FUNCTION_BLOCK handle
VAR_INPUT
END_VAR
VAR_OUTPUT
END_VAR
VAR
	i,j,k:INT;
	v_step		: LREAL;
	avg_window	: INT;
	avg_window_size : INT := 20;
	return_handoff_bypass : BOOL;

	act_hh		:	ARRAY[1..7] OF ARRAY [1..30] OF LREAL;
	pos_abs		:	LREAL;
	legacy_vel	:	LREAL;

	init_done : BOOL := FALSE;
	all_enabled : BOOL;
	all_powered : BOOL;
	has_axis_error : BOOL;
	hold_active : BOOL := FALSE;

	// 上位机通信看门狗。超时锁存后只能通过显式恢复握手解除。
	host_watchdog_timer : TON;
	host_last_session_id : UDINT := 0;
	host_last_heartbeat_sequence : UDINT := 0;
	host_heartbeat_seen : BOOL := FALSE;
	host_session_changed : BOOL;
	host_heartbeat_changed : BOOL;
	host_timeout_latched : BOOL := TRUE;
	host_timeout_prev : BOOL := FALSE;
	// 看门狗超时后锁存一次外部设定值保持位置。
	// 不能每拍把 Actual Position 回写为下一拍设定值，否则编码器微动会被回灌到 NC。
	host_hold_abs : ARRAY[1..7] OF LREAL;
	host_hold_captured : BOOL := FALSE;
	host_all_stopped : BOOL;
	host_return_stop_active : ARRAY[1..7] OF BOOL;
	host_return_stop_exec : ARRAY[1..7] OF BOOL;
	host_axis4_stop_active : BOOL := FALSE;
	fb_host_return_stop : ARRAY[1..7] OF MC_Stop;

	right_slimit : ARRAY[1..7] OF LREAL;
	rslimit_distance	: ARRAY[1..7] OF LREAL := [99.0, 0.0, 666.0, 0.0, 688.0, 688.0, 0.0];
	slimit_enable : ARRAY[1..7] OF BOOL := [TRUE, FALSE, FALSE, FALSE, TRUE, TRUE, FALSE];

	ext_setpoint_enabled : ARRAY[1..7] OF BOOL := [FALSE,FALSE,FALSE,FALSE,FALSE,FALSE,FALSE];
	spg_enable_exec	: ARRAY[1..7] OF BOOL;
	spg_disable_exec : ARRAY[1..7] OF BOOL;

	return_enable : ARRAY[1..7] OF BOOL := [TRUE, FALSE, FALSE, FALSE, TRUE, TRUE, FALSE];
	return_state : ARRAY[1..7] OF INT;
	return_exec : ARRAY[1..7] OF BOOL;
	return_target_abs : ARRAY[1..7] OF LREAL;
	return_velocity : ARRAY[1..7] OF LREAL;
	return_acc : ARRAY[1..7] OF LREAL;
	return_dec : ARRAY[1..7] OF LREAL;
	return_jerk : ARRAY[1..7] OF LREAL;
	return_finish_error : ARRAY[1..7] OF BOOL;
	return_cancelled : ARRAY[1..7] OF BOOL;
	return_error_id_pending : ARRAY[1..7] OF UDINT;
	fb_return_move_abs : ARRAY[1..7] OF MC_MoveAbsolute;

	axis4_manual_state : INT := 0;
	axis4_request_dir_now : INT := 0;
	axis4_requested_dir : INT := 0;
	axis4_pending_dir : INT := 0;
	axis4_move_exec : BOOL := FALSE;
	axis4_stop_exec : BOOL := FALSE;
	axis4_finish_error : BOOL := FALSE;
	axis4_error_id_pending : UDINT := 0;
	axis4_manual_velocity : LREAL := 30;
	axis4_manual_acc : LREAL := 100;
	axis4_manual_dec : LREAL := 100;
	axis4_manual_jerk : LREAL := 500.0;
	axis4_manual_direction : MC_Direction := MC_Direction.MC_Positive_Direction;
	fb_axis4_move_velocity : MC_MoveVelocity;
	fb_axis4_stop : MC_Stop;
	ramp_counter: ARRAY[1..7] OF INT;
	act_h_prev : ARRAY[1..7] OF LREAL;

	traj_pos     : ARRAY[1..7] OF LREAL;
	traj_vel     : ARRAY[1..7] OF LREAL;
	traj_acc     : ARRAY[1..7] OF LREAL;
	acc_raw      : LREAL;

	traj_wn      : LREAL := 60.0;
	traj_vmax    : ARRAY[1..7] OF LREAL := [80, 0, 0, 0, 80, 80, 0];
	traj_amax    : ARRAY[1..7] OF LREAL := [2000, 0, 0, 0, 2000, 2000, 0];
	traj_enable  : ARRAY[1..7] OF BOOL := [TRUE, FALSE, FALSE, FALSE, TRUE, TRUE, FALSE];
	pd_mode : USINT;
	pd_state : USINT;
	pd_last_state : USINT;
	pd_last_sync : USINT;
	pd_step : USINT;
	pd_axis : INT := 1;
	pd_active : ARRAY[1..7] OF BOOL;
	pd_req : ARRAY[1..7] OF BOOL;
	pd_moved : ARRAY[1..7] OF BOOL;
	pd_ref : ARRAY[1..7] OF LREAL;
	pd_target : ARRAY[1..7] OF LREAL;
	pd_forward : ST_AxisPlannedReturnCmd;
	pd_return : ST_AxisPlannedReturnCmd;
	pd_release_wait, pd_reclamp_wait, pd_release_lead, pd_reclamp_lead : TIME;
	pd_open2, pd_close2, pd_open4, pd_close4 : WORD;
	pd_coupling : BOOL;
	pd_ready : BOOL;
	pd_fault : BOOL;
	pd_all_done : BOOL;
	pd_anchor1, pd_anchor5, pd_anchor6, pd_input1, pd_input2 : LREAL;
	pd_baseline_timer, pd_release_timer, pd_reclamp_timer : TON;
	pd_release_lead_timer, pd_reclamp_lead_timer : TON;
	rec_block : INT := 1;
	rec_index : INT;
	rec_sample : UDINT;
	rec_sequence : UDINT;
	rec_was_active : BOOL;
	rec_capture : BOOL;
	rec_time : ULINT;
	zero_index : UINT;
	zero_force, zero_sum, zero_square, zero_mean, zero_std : ARRAY[1..4] OF LREAL;
END_VAR

host_session_changed := G.host_session_id <> host_last_session_id;
host_heartbeat_changed := host_session_changed OR
	(G.host_heartbeat_sequence <> host_last_heartbeat_sequence);

IF host_session_changed THEN
	// 非零会话发生变化表示新的上位机接管，必须重新完成恢复握手。
	IF host_last_session_id <> 0 THEN
		host_timeout_latched := TRUE;
	END_IF
	host_last_session_id := G.host_session_id;
END_IF

IF host_heartbeat_changed THEN
	host_last_heartbeat_sequence := G.host_heartbeat_sequence;
END_IF

host_heartbeat_seen := G.host_session_id <> 0;
// 心跳变化的扫描周期将 TON 复位；序号连续 100 ms 不变化才判定通信超时。
host_watchdog_timer(
	IN:=host_heartbeat_seen AND NOT host_heartbeat_changed,
	PT:=T#100MS
);
IF (NOT host_heartbeat_seen) OR host_watchdog_timer.Q THEN
	host_timeout_latched := TRUE;
END_IF
G.host_comm_timeout := host_timeout_latched;

IF G.handle_reinit_req THEN
	init_done := FALSE;
	G.handle_reinit_done := FALSE;
	G.handle_reinit_req := FALSE;
	G.estop_hold_req := TRUE;

	FOR i:=1 TO 7 DO
		ext_setpoint_enabled[i] := FALSE;
		spg_enable_exec[i] := FALSE;
		spg_disable_exec[i] := FALSE;
		return_state[i] := 0;
		return_exec[i] := FALSE;
		return_finish_error[i] := FALSE;
		return_cancelled[i] := FALSE;
		return_error_id_pending[i] := 0;
		host_return_stop_active[i] := FALSE;
		host_return_stop_exec[i] := FALSE;
		traj_pos[i] := 0.0;
		traj_vel[i] := 0.0;
		traj_acc[i] := 0.0;
		host_hold_abs[i] := 0.0;
		G.return_cmd[i].Req := FALSE;
		G.return_cmd[i].Busy := FALSE;
		G.return_cmd[i].Done := FALSE;
		G.return_cmd[i].Error := FALSE;
		G.return_cmd[i].ErrorId := 0;
	END_FOR
	host_hold_captured := FALSE;
	host_timeout_prev := FALSE;

	axis4_manual_state := 0;
	axis4_request_dir_now := 0;
	axis4_requested_dir := 0;
	axis4_pending_dir := 0;
	axis4_move_exec := FALSE;
	axis4_stop_exec := FALSE;
	axis4_finish_error := FALSE;
	axis4_error_id_pending := 0;
	G.axis4_fwd_req := FALSE;
	G.axis4_rev_req := FALSE;
	G.axis4_manual_busy := FALSE;
	G.axis4_manual_done := FALSE;
	G.axis4_manual_error := FALSE;
	G.axis4_manual_error_id := 0;
END_IF

IF NOT init_done THEN
	G.estop_hold_req := TRUE;
	G.power_[3].Enable := FALSE;
	all_enabled := TRUE;
	FOR i:=1 TO 7 DO
		IF i = 3 THEN
			G.SetPointGenEnable[i](Axis:=G.axis[i], Execute:=FALSE);
		ELSE
			G.SetPointGenEnable[i](Axis:=G.axis[i], Execute:=TRUE);
			IF NOT G.SetPointGenEnable[i].Done THEN
				all_enabled := FALSE;
			END_IF
		END_IF
	END_FOR
	
	IF all_enabled THEN
		FOR j:=1 TO 7 DO
			G.Act_pos[j] := G.axis[j].NcToPlc.ActPos - G.init_pos[j];
			G.act_pos_from_left[j] := G.axis[j].NcToPlc.ActPos - G.leftlimit[j];
			G.ref_slow[j] := G.Act_pos[j];
			G.act_h[j] := G.Act_pos[j];
			G.act_hf[j] := G.Act_pos[j];
			G.refer[j] := G.Act_pos[j];
			G.refer_from_left[j] := G.act_pos_from_left[j];
			ext_setpoint_enabled[j] := j <> 3;

			FOR k:=1 TO 30 DO
				act_hh[j][k] := G.Act_pos[j];
			END_FOR
			act_h_prev[j] := G.Act_pos[j];
			traj_pos[j] := G.Act_pos[j];
			traj_vel[j] := 0.0;
			traj_acc[j] := 0.0;
			IF slimit_enable[j] THEN
				right_slimit[j] := G.leftlimit[j] + rslimit_distance[j];
			END_IF
			G.return_cmd[j].Busy := FALSE;
			G.return_cmd[j].Done := FALSE;
			G.return_cmd[j].Error := FALSE;
			G.return_cmd[j].ErrorId := 0;
		END_FOR

		G.axis4_manual_busy := FALSE;
		G.axis4_manual_done := FALSE;
		G.axis4_manual_error := FALSE;
		G.axis4_manual_error_id := 0;

		init_done := TRUE;
		// 通信超时未解除时不提前确认恢复；正式握手后会再次进入本初始化流程。
		G.handle_reinit_done := NOT G.host_comm_timeout;
	END_IF
	RETURN;
END_IF

G.estop_hold_req := FALSE;
G.power_[3].Enable := FALSE;
G.power_[5].Enable := TRUE;

all_powered := TRUE;
FOR i:=1 TO 7 DO
	IF i <> 3 AND NOT (G.program_test_mode = 1 AND i = 5) AND NOT G.power_output[i].Done THEN
		all_powered := FALSE;
		EXIT;
	END_IF
END_FOR

has_axis_error := FALSE;
FOR i:=1 TO 7 DO
	IF i = 3 OR (G.program_test_mode = 1 AND i = 5) THEN
		CONTINUE;
	END_IF
	IF G.axis[i].Status.Error OR G.power_output[i].Error OR G.reset_output[i].Error THEN
		has_axis_error := TRUE;
		EXIT;
	END_IF
END_FOR


IF (NOT all_powered) OR has_axis_error OR G.host_comm_timeout THEN
	pd_fault := TRUE;
	ProgramDelivery();
	ProgramRecord();
END_IF

IF NOT all_powered THEN
	G.estop_hold_req := TRUE;
	hold_active := TRUE;
	FOR j:=1 TO 7 DO
		G.Act_pos[j] := G.axis[j].NcToPlc.ActPos - G.init_pos[j];
		G.act_pos_from_left[j] := G.axis[j].NcToPlc.ActPos - G.leftlimit[j];
		G.refer[j] := G.Act_pos[j];
		G.ref_slow[j] := G.Act_pos[j];
		G.act_h[j] := G.Act_pos[j];
		G.act_hf[j] := G.Act_pos[j];
		G.refer_from_left[j] := G.act_pos_from_left[j];
		FOR k:=1 TO 30 DO
			act_hh[j][k] := G.Act_pos[j];
		END_FOR
		act_h_prev[j] := G.Act_pos[j];
		traj_pos[j] := G.Act_pos[j];
		traj_vel[j] := 0.0;
		traj_acc[j] := 0.0;
	END_FOR
	IF has_axis_error THEN
		G.gen_state := _err;
	END_IF
	RETURN;
END_IF

IF hold_active THEN
	hold_active := FALSE;
	G.handle_reinit_req := TRUE;
	G.estop_hold_req := TRUE;
	IF has_axis_error THEN
		G.gen_state := _err;
	END_IF
	RETURN;
END_IF

IF has_axis_error THEN
	G.estop_hold_req := TRUE;
	G.gen_state := _err;
	RETURN;
END_IF

IF G.host_comm_timeout THEN
	G.estop_hold_req := TRUE;
	G.handle_reinit_done := FALSE;

	IF (NOT host_timeout_prev) OR (NOT host_hold_captured) THEN
		// 仅在进入超时保持时采样一次。之后始终维持同一绝对位置，
		// 避免 Actual -> Set Position 的逐周期回灌导致低频来回摆动。
		FOR i:=1 TO 7 DO
			host_hold_abs[i] := G.axis[i].NcToPlc.ActPos;
		END_FOR
		host_hold_captured := TRUE;
	END_IF

	IF NOT host_timeout_prev THEN
		// 仅捕获超时发生时已经在运行的独立运动，禁止恢复后自动续跑。
		FOR i:=1 TO 7 DO
			host_return_stop_active[i] :=
				(return_state[i] <> 0) OR G.return_cmd[i].Busy OR fb_return_move_abs[i].Busy;
			host_return_stop_exec[i] := FALSE;
		END_FOR
		host_axis4_stop_active := (axis4_manual_state <> 0) OR fb_axis4_move_velocity.Busy;
	END_IF

	// 超时期间持续清除运动请求，避免上位机重连时把旧请求重新送入状态机。
	G.axis1_fast_return := FALSE;
	G.axis6_fast_retract := FALSE;
	G.axis4_fwd_req := FALSE;
	G.axis4_rev_req := FALSE;
	G.startup_smoothing_bypass := FALSE;
	axis4_move_exec := FALSE;
	host_all_stopped := TRUE;

	FOR i:=1 TO 7 DO
		spg_enable_exec[i] := FALSE;
		spg_disable_exec[i] := FALSE;
		return_exec[i] := FALSE;
		G.return_cmd[i].Req := FALSE;
		G.return_cmd[i].Done := FALSE;

		// 实际位置仍实时刷新用于诊断；外部参考始终保持超时边沿的锁存位置。
		G.Act_pos[i] := G.axis[i].NcToPlc.ActPos - G.init_pos[i];
		G.act_pos_from_left[i] := G.axis[i].NcToPlc.ActPos - G.leftlimit[i];
		G.refer[i] := host_hold_abs[i] - G.init_pos[i];
		G.ref_slow[i] := G.refer[i];
		G.act_h[i] := G.refer[i];
		G.act_hf[i] := G.refer[i];
		G.refer_from_left[i] := host_hold_abs[i] - G.leftlimit[i];
		FOR k:=1 TO 30 DO
			act_hh[i][k] := G.refer[i];
		END_FOR
		act_h_prev[i] := G.refer[i];
		traj_pos[i] := G.refer[i];
		traj_vel[i] := 0.0;
		traj_acc[i] := 0.0;

		IF host_return_stop_active[i] THEN
			IF fb_host_return_stop[i].Done THEN
				host_return_stop_exec[i] := FALSE;
				host_return_stop_active[i] := FALSE;
			ELSIF fb_host_return_stop[i].Error THEN
				// 拉低一个扫描周期清除错误，下一周期继续尝试受控停止。
				host_return_stop_exec[i] := FALSE;
				host_all_stopped := FALSE;
			ELSE
				host_return_stop_exec[i] := TRUE;
				host_all_stopped := FALSE;
			END_IF
		ELSE
			host_return_stop_exec[i] := FALSE;
		END_IF
		G.return_cmd[i].Busy := host_return_stop_active[i];

		IF ext_setpoint_enabled[i] THEN
			MC_ExtSetPointGenFeed(
				Position:=host_hold_abs[i],
				Velocity:=0.0,
				Acceleration:=0.0,
				Direction:=1,
				Axis:=G.axis[i]);
		END_IF

		// 所有运动功能块在看门狗分支中仍保持每扫描调用。
		G.SetPointGenEnable[i](Axis:=G.axis[i], Execute:=FALSE);
		G.SetPointGenDisable[i](Axis:=G.axis[i], Execute:=FALSE);
		fb_return_move_abs[i](
			Axis:=G.axis[i],
			Position:=return_target_abs[i],
			Velocity:=return_velocity[i],
			Acceleration:=return_acc[i],
			Deceleration:=return_dec[i],
			Jerk:=return_jerk[i],
			Execute:=FALSE
		);
		fb_host_return_stop[i](
			Axis:=G.axis[i],
			Execute:=host_return_stop_exec[i],
			Deceleration:=100.0,
			Jerk:=500.0
		);
	END_FOR

	IF host_axis4_stop_active THEN
		IF fb_axis4_stop.Done THEN
			axis4_stop_exec := FALSE;
			host_axis4_stop_active := FALSE;
		ELSIF fb_axis4_stop.Error THEN
			// 拉低一个扫描周期清除错误，下一周期继续尝试受控停止。
			axis4_stop_exec := FALSE;
			host_all_stopped := FALSE;
		ELSE
			axis4_stop_exec := TRUE;
			host_all_stopped := FALSE;
		END_IF
	ELSE
		axis4_stop_exec := FALSE;
	END_IF
	G.axis4_manual_busy := host_axis4_stop_active;
	G.axis4_manual_done := FALSE;

	fb_axis4_move_velocity(
		Axis:=G.axis[4],
		Execute:=FALSE,
		Velocity:=axis4_manual_velocity,
		Acceleration:=axis4_manual_acc,
		Deceleration:=axis4_manual_dec,
		Jerk:=axis4_manual_jerk,
		Direction:=axis4_manual_direction
	);
	fb_axis4_stop(
		Axis:=G.axis[4],
		Execute:=axis4_stop_exec,
		Deceleration:=axis4_manual_dec,
		Jerk:=axis4_manual_jerk
	);

	// 清请求并解除超时即为 PLC 对恢复请求的确认；随后复用既有重初始化流程。
	IF G.host_recover_req AND host_heartbeat_seen AND
		(NOT host_watchdog_timer.Q) AND host_all_stopped THEN
		host_timeout_latched := FALSE;
		G.host_comm_timeout := FALSE;
		G.host_recover_req := FALSE;
		G.handle_reinit_req := TRUE;
	END_IF

	host_timeout_prev := G.host_comm_timeout;
	RETURN;
END_IF

host_timeout_prev := FALSE;
host_hold_captured := FALSE;
// 非超时状态收到的恢复请求没有业务含义，清除以免成为下一次超时的陈旧握手。
G.host_recover_req := FALSE;

pd_fault := FALSE;
ProgramDelivery();
ProgramRecord();

IF G.cylinder5_press_req THEN
	G.cylinder5_value := 0;
ELSE
	G.cylinder5_value := 2000;
END_IF

FOR i:=1 TO 7 DO
	spg_enable_exec[i] := FALSE;
	spg_disable_exec[i] := FALSE;
	return_exec[i] := FALSE;
END_FOR
axis4_move_exec := FALSE;
axis4_stop_exec := FALSE;

FOR j:=1 TO 7 DO
	G.Act_pos[j] := G.axis[j].NcToPlc.ActPos - G.init_pos[j];
	G.act_pos_from_left[j] := G.axis[j].NcToPlc.ActPos - G.leftlimit[j];
	G.refer_from_left[j] := (G.refer[j] + G.init_pos[j]) - G.leftlimit[j];

	v_step := G.v_limit[j];
	// 回退接管旁路：回退 Busy 期间跳过斜坡/均值，避免回退末端重新进入慢链路
	return_handoff_bypass := ((j = 1) AND (G.axis1_fast_return OR G.return_cmd[1].Busy))
		OR ((j = 6) AND (G.axis6_fast_retract OR G.return_cmd[6].Busy));
	IF return_handoff_bypass THEN
		avg_window := 1;
		ramp_counter[j] := 0;
	ELSE
		ramp_counter[j] := MIN(ramp_counter[j] + 1, avg_window_size);
		avg_window := MAX(1, ramp_counter[j]);
	END_IF

	FOR k:=2 TO 20 DO
		act_hh[j][22-k] := act_hh[j][21-k];
	END_FOR

	IF slimit_enable[j] THEN
		IF (G.axis[j].NcToPlc.ActPos >= right_slimit[j]) AND (G.refer[j] > G.ref_slow[j]) THEN
			G.refer[j] := G.ref_slow[j];
		END_IF
	END_IF

	IF return_handoff_bypass THEN
		G.ref_slow[j] := G.refer[j];
	ELSIF (G.refer[j] - G.ref_slow[j]) > v_step THEN
		G.ref_slow[j] := G.ref_slow[j] + v_step;
	ELSIF (G.refer[j] - G.ref_slow[j]) < -v_step THEN
		G.ref_slow[j] := G.ref_slow[j] - v_step;
	ELSE
		G.ref_slow[j] := G.refer[j];
	END_IF

	IF return_handoff_bypass THEN
		FOR i:=1 TO 20 DO
			act_hh[j][i] := G.ref_slow[j];
		END_FOR
		G.act_h[j] := G.ref_slow[j];
	ELSE
		act_hh[j][1] := G.ref_slow[j];
		G.act_h[j] := 0;
		FOR i:=1 TO avg_window DO
			G.act_h[j] := G.act_h[j] + act_hh[j][i] / TO_LREAL(avg_window);
		END_FOR
	END_IF

	IF traj_enable[j] AND NOT return_handoff_bypass AND NOT G.startup_smoothing_bypass THEN
		acc_raw := traj_wn * traj_wn * (G.refer[j] - traj_pos[j]) - 2.0 * traj_wn * traj_vel[j];
		IF acc_raw > traj_amax[j] THEN
			acc_raw := traj_amax[j];
		ELSIF acc_raw < -traj_amax[j] THEN
			acc_raw := -traj_amax[j];
		END_IF
		traj_acc[j] := acc_raw;
		traj_vel[j] := traj_vel[j] + 0.001 * traj_acc[j];
		IF traj_vel[j] > traj_vmax[j] THEN
			traj_vel[j] := traj_vmax[j];
		ELSIF traj_vel[j] < -traj_vmax[j] THEN
			traj_vel[j] := -traj_vmax[j];
		END_IF
		traj_pos[j] := traj_pos[j] + 0.001 * traj_vel[j];
		IF ABS(G.refer[j] - traj_pos[j]) < 0.001 AND ABS(traj_vel[j]) < 0.01 THEN
			traj_pos[j] := G.refer[j];
			traj_vel[j] := 0.0;
			traj_acc[j] := 0.0;
		END_IF
	ELSE
		traj_pos[j] := G.act_h[j];
		traj_vel[j] := 0.0;
		traj_acc[j] := 0.0;
	END_IF
END_FOR

FOR i:=1 TO 7 DO
	IF NOT return_enable[i] AND NOT ((pd_mode <> 0) AND ((i = 2) OR (i = 7))) THEN
		CONTINUE;
	END_IF

	IF return_state[i] = 0 THEN
		G.return_cmd[i].Busy := FALSE;
		host_return_stop_active[i] := FALSE;
		host_return_stop_exec[i] := FALSE;
		IF NOT G.return_cmd[i].Req THEN
			G.return_cmd[i].Done := FALSE;
			G.return_cmd[i].Error := FALSE;
			G.return_cmd[i].ErrorId := 0;
			return_finish_error[i] := FALSE;
			return_cancelled[i] := FALSE;
			return_error_id_pending[i] := 0;
		ELSIF (NOT G.return_cmd[i].Done) AND (NOT G.return_cmd[i].Error) THEN
			// Req 由上位机在完整写入参数后最后置位；此处只锁存一次，
			// 本次 MC_MoveAbsolute 后续不再直接读取可被 ADS 改写的命令参数。
			return_target_abs[i] := G.return_cmd[i].TargetAbs;
			return_velocity[i] := G.return_cmd[i].Velocity;
			return_acc[i] := G.return_cmd[i].Acc;
			return_dec[i] := G.return_cmd[i].Dec;
			return_jerk[i] := G.return_cmd[i].Jerk;
			return_cancelled[i] := FALSE;
			return_state[i] := 10;
		END_IF
	END_IF

	// 上位机在任何尚未完成的阶段撤销请求时，都先受控停止轴。
	// return_cancelled防止状态40复用30/31收尾后因Req仍为FALSE再次进入停止环。
	IF ((return_state[i] = 10) OR (return_state[i] = 20) OR
		(return_state[i] = 30) OR (return_state[i] = 31)) AND
		(NOT G.return_cmd[i].Req) AND (NOT return_cancelled[i]) THEN
		return_exec[i] := FALSE;
		spg_enable_exec[i] := FALSE;
		spg_disable_exec[i] := FALSE;
		return_cancelled[i] := TRUE;
		host_return_stop_active[i] := TRUE;
		// 清除上一次执行沿；状态 40 首次处理时不会采信旧的 Done/Error。
		host_return_stop_exec[i] := FALSE;
		G.return_cmd[i].Done := FALSE;
		G.return_cmd[i].Error := FALSE;
		G.return_cmd[i].ErrorId := 0;
		return_state[i] := 40;
	END_IF

	CASE return_state[i] OF
	10:
		G.return_cmd[i].Busy := TRUE;
		spg_disable_exec[i] := TRUE;
		IF G.SetPointGenDisable[i].Done OR NOT G.SetPointGenDisable[i].Enabled THEN
			ext_setpoint_enabled[i] := FALSE;
			return_state[i] := 20;
		END_IF

	20:
		G.return_cmd[i].Busy := TRUE;
		return_exec[i] := TRUE;
		G.refer_from_left[i] := return_target_abs[i] - G.leftlimit[i];

		IF fb_return_move_abs[i].Done OR
		   ((NOT fb_return_move_abs[i].Busy) AND (ABS(G.axis[i].NcToPlc.ActPos - return_target_abs[i]) <= 0.05)) THEN
			return_finish_error[i] := FALSE;
			return_error_id_pending[i] := 0;
			return_state[i] := 30;
		ELSIF fb_return_move_abs[i].Error OR fb_return_move_abs[i].CommandAborted THEN
			return_finish_error[i] := TRUE;
			return_error_id_pending[i] := fb_return_move_abs[i].ErrorID;
			return_state[i] := 30;
		END_IF

	30:
		G.return_cmd[i].Busy := TRUE;
		IF ABS(G.axis[i].NcToPlc.ActVelo) <= 0.5 THEN
			G.Act_pos[i] := G.axis[i].NcToPlc.ActPos - G.init_pos[i];
			G.act_pos_from_left[i] := G.axis[i].NcToPlc.ActPos - G.leftlimit[i];
			G.refer[i] := G.Act_pos[i];
			G.ref_slow[i] := G.Act_pos[i];
			G.act_h[i] := G.Act_pos[i];
			G.act_hf[i] := G.Act_pos[i];
			G.refer_from_left[i] := G.act_pos_from_left[i];
			FOR k:=1 TO 30 DO
				act_hh[i][k] := G.Act_pos[i];
			END_FOR
			act_h_prev[i] := G.Act_pos[i];
			traj_pos[i] := G.Act_pos[i];
			traj_vel[i] := 0.0;
			traj_acc[i] := 0.0;
			// 先留出一个完整 PLC 扫描周期预送当前设定值，再重新使能外部设定值发生器。
			return_state[i] := 31;
		END_IF

	31:
		G.return_cmd[i].Busy := TRUE;
		spg_enable_exec[i] := TRUE;
		IF G.SetPointGenEnable[i].Done THEN
			ext_setpoint_enabled[i] := TRUE;
			G.return_cmd[i].Busy := FALSE;
			IF return_finish_error[i] THEN
				G.return_cmd[i].Done := FALSE;
				G.return_cmd[i].Error := TRUE;
				G.return_cmd[i].ErrorId := return_error_id_pending[i];
			ELSIF return_cancelled[i] THEN
				// 主动取消只表示已经安全停稳，不把取消伪装成原计划动作成功完成。
				G.return_cmd[i].Done := FALSE;
				G.return_cmd[i].Error := FALSE;
				G.return_cmd[i].ErrorId := 0;
			ELSE
				G.return_cmd[i].Done := TRUE;
				G.return_cmd[i].Error := FALSE;
				G.return_cmd[i].ErrorId := 0;
			END_IF
			return_finish_error[i] := FALSE;
			return_cancelled[i] := FALSE;
			return_error_id_pending[i] := 0;
			return_state[i] := 0;
		END_IF

	40:
		G.return_cmd[i].Busy := TRUE;
		G.return_cmd[i].Done := FALSE;
		return_exec[i] := FALSE;
		spg_enable_exec[i] := FALSE;
		spg_disable_exec[i] := FALSE;
		// 状态40仍以实际停稳为退出条件。若原运动或此前的MC_Stop已经报错，
		// 在继续受控停止期间保持错误对上位机可见，不能用Busy掩盖故障。
		IF return_finish_error[i] THEN
			G.return_cmd[i].Error := TRUE;
			G.return_cmd[i].ErrorId := return_error_id_pending[i];
		END_IF

		IF host_return_stop_exec[i] THEN
			IF fb_host_return_stop[i].Done THEN
				// 停稳后释放 MC_Stop，并复用状态 30/31 按实际位置重建和恢复外部设定值。
				host_return_stop_exec[i] := FALSE;
				host_return_stop_active[i] := FALSE;
				return_state[i] := 30;
			ELSIF fb_host_return_stop[i].Error THEN
				// 原运动错误优先；否则锁存首次MC_Stop错误并立即通知上位机。
				// Busy和停止任务保持有效，Execute拉低一拍后仍继续尝试受控停止，
				// 只有真实Done才能进入位置重建，绝不把停止失败伪装成完成。
				IF NOT return_finish_error[i] THEN
					return_finish_error[i] := TRUE;
					return_error_id_pending[i] := fb_host_return_stop[i].ErrorID;
				END_IF
				G.return_cmd[i].Error := TRUE;
				G.return_cmd[i].ErrorId := return_error_id_pending[i];
				host_return_stop_exec[i] := FALSE;
			END_IF
		ELSIF NOT fb_host_return_stop[i].Error THEN
			// 首次进入或错误已由低电平清除后，启动（或重试）受控停止。
			host_return_stop_exec[i] := TRUE;
		END_IF
	END_CASE
END_FOR

axis4_request_dir_now := 0;
IF G.axis4_fwd_req AND NOT G.axis4_rev_req THEN
	axis4_request_dir_now := 1;
ELSIF G.axis4_rev_req AND NOT G.axis4_fwd_req THEN
	axis4_request_dir_now := -1;
END_IF

IF axis4_manual_state = 0 THEN
	G.axis4_manual_busy := FALSE;
	IF axis4_request_dir_now = 0 THEN
		G.axis4_manual_done := FALSE;
		G.axis4_manual_error := FALSE;
		G.axis4_manual_error_id := 0;
	ELSIF NOT G.axis4_manual_error THEN
		G.axis4_manual_done := FALSE;
		G.axis4_manual_error := FALSE;
		G.axis4_manual_error_id := 0;
		axis4_requested_dir := axis4_request_dir_now;
		axis4_pending_dir := 0;
		axis4_finish_error := FALSE;
		axis4_error_id_pending := 0;
		axis4_manual_state := 10;
	END_IF
END_IF

CASE axis4_manual_state OF
10:
	G.axis4_manual_busy := TRUE;
	spg_disable_exec[4] := TRUE;
	IF G.SetPointGenDisable[4].Done OR NOT G.SetPointGenDisable[4].Enabled THEN
		ext_setpoint_enabled[4] := FALSE;
		axis4_manual_state := 20;
	END_IF

20:
	G.axis4_manual_busy := TRUE;
	axis4_pending_dir := axis4_request_dir_now;
	IF axis4_requested_dir >= 0 THEN
		axis4_manual_direction := MC_Direction.MC_Positive_Direction;
	ELSE
		axis4_manual_direction := MC_Direction.MC_Negative_Direction;
	END_IF

	IF axis4_pending_dir = 0 THEN
		axis4_manual_state := 30;
	ELSIF axis4_pending_dir <> axis4_requested_dir THEN
		axis4_manual_state := 30;
	ELSE
		axis4_move_exec := TRUE;
	END_IF

	IF fb_axis4_move_velocity.Error OR fb_axis4_move_velocity.CommandAborted THEN
		axis4_finish_error := TRUE;
		axis4_error_id_pending := fb_axis4_move_velocity.ErrorID;
		G.axis4_manual_error_id := fb_axis4_move_velocity.ErrorID;
		axis4_pending_dir := 0;
		axis4_manual_state := 40;
	END_IF

30:
	G.axis4_manual_busy := TRUE;
	axis4_pending_dir := axis4_request_dir_now;
	axis4_stop_exec := TRUE;

	IF fb_axis4_stop.Error THEN
		axis4_finish_error := TRUE;
		axis4_error_id_pending := fb_axis4_stop.ErrorID;
		axis4_pending_dir := 0;
		axis4_manual_state := 39;
	ELSIF fb_axis4_stop.Done OR (ABS(G.axis[4].NcToPlc.ActVelo) <= 0.05) THEN
		IF axis4_pending_dir <> 0 THEN
			axis4_requested_dir := axis4_pending_dir;
			axis4_manual_state := 20;
		ELSE
			axis4_requested_dir := 0;
			axis4_manual_state := 39;
		END_IF
	END_IF

39:
G.axis4_manual_busy := TRUE;
// MC_Stop needs one cycle with Execute=FALSE before SetPointGenEnable can get a clean rising edge
axis4_manual_state := 40;
	
40:
	G.axis4_manual_busy := TRUE;
	G.Act_pos[4] := G.axis[4].NcToPlc.ActPos - G.init_pos[4];
	G.act_pos_from_left[4] := G.axis[4].NcToPlc.ActPos - G.leftlimit[4];
	G.refer[4] := G.Act_pos[4];
	G.ref_slow[4] := G.Act_pos[4];
	G.act_h[4] := G.Act_pos[4];
	G.act_hf[4] := G.Act_pos[4];
	G.refer_from_left[4] := G.act_pos_from_left[4];
	FOR k:=1 TO 30 DO
		act_hh[4][k] := G.Act_pos[4];
	END_FOR
	act_h_prev[4] := G.Act_pos[4];
	traj_pos[4] := G.Act_pos[4];
	traj_vel[4] := 0.0;
	traj_acc[4] := 0.0;
	spg_enable_exec[4] := TRUE;
	IF G.SetPointGenEnable[4].Done THEN
		ext_setpoint_enabled[4] := TRUE;
		G.axis4_manual_busy := FALSE;
		IF axis4_finish_error THEN
			G.axis4_manual_done := FALSE;
			G.axis4_manual_error := TRUE;
			G.axis4_manual_error_id := axis4_error_id_pending;
		ELSE
			G.axis4_manual_done := TRUE;
			G.axis4_manual_error := FALSE;
			G.axis4_manual_error_id := 0;
		END_IF
		axis4_finish_error := FALSE;
		axis4_error_id_pending := 0;
		axis4_manual_state := 0;
	END_IF
END_CASE

FOR i:=1 TO 7 DO
	IF i <> 3 AND G.power_output[i].Error THEN
		G.axis_Reset[i].Execute := TRUE;
	END_IF
END_FOR

FOR i:=1 TO 7 DO
	IF i = 3 THEN
		G.act_hf[i] := G.axis[i].NcToPlc.ActPos - G.init_pos[i];
	ELSIF ext_setpoint_enabled[i] OR (return_state[i] = 31) OR spg_enable_exec[i] THEN
		IF traj_enable[i] AND NOT G.startup_smoothing_bypass THEN
			pos_abs := traj_pos[i] + G.init_pos[i];
			MC_ExtSetPointGenFeed(
				Position     := pos_abs,
				Velocity     := traj_vel[i],
				Acceleration := traj_acc[i],
				Direction    := 1,
				Axis         := G.axis[i]);
		ELSE
			pos_abs := G.act_h[i] + G.init_pos[i];
			legacy_vel := (G.act_h[i] - act_h_prev[i]) / 0.001;
			MC_ExtSetPointGenFeed(
				Position     := pos_abs,
				Velocity     := legacy_vel,
				Acceleration := 0,
				Direction    := 1,
				Axis         := G.axis[i]);
		END_IF
		G.act_hf[i] := G.act_h[i];
	ELSE
		G.act_hf[i] := G.axis[i].NcToPlc.ActPos - G.init_pos[i];
	END_IF
	act_h_prev[i] := G.act_h[i];
END_FOR

FOR i:=1 TO 7 DO
	G.SetPointGenEnable[i](Axis:=G.axis[i], Execute:=spg_enable_exec[i]);
	G.SetPointGenDisable[i](Axis:=G.axis[i], Execute:=spg_disable_exec[i]);
	fb_return_move_abs[i](
		Axis:=G.axis[i],
		Position:=return_target_abs[i],
		Velocity:=return_velocity[i],
		Acceleration:=return_acc[i],
		Deceleration:=return_dec[i],
		Jerk:=return_jerk[i],
		Execute:=return_exec[i]
	);
	fb_host_return_stop[i](
		Axis:=G.axis[i],
		Execute:=host_return_stop_exec[i],
		Deceleration:=100.0,
		Jerk:=500.0
	);
END_FOR

fb_axis4_move_velocity(
	Axis:=G.axis[4],
	Execute:=axis4_move_exec,
	Velocity:=axis4_manual_velocity,
	Acceleration:=axis4_manual_acc,
	Deceleration:=axis4_manual_dec,
	Jerk:=axis4_manual_jerk,
	Direction:=axis4_manual_direction
);
fb_axis4_stop(
	Axis:=G.axis[4],
	Execute:=axis4_stop_exec,
	Deceleration:=axis4_manual_dec,
	Jerk:=axis4_manual_jerk
);

ACTION ProgramDelivery:


pd_all_done := TRUE;
FOR i := 1 TO 7 DO
	IF (return_state[i] <> 0) OR G.return_cmd[i].Busy THEN pd_all_done := FALSE; END_IF
END_FOR
IF G.program_test_mode <> pd_mode THEN
	IF ((pd_state = 0) OR (pd_state >= 10)) AND NOT G.program_test_setup_busy AND pd_all_done THEN
		pd_mode := G.program_test_mode;
		pd_state := 0;
		pd_step := 0;
		pd_ready := FALSE;
		G.program_test_setup_done := FALSE;
		G.program_test_status_error_id := 0;
		G.program_test_handle_cycle := 0;
		FOR i := 1 TO 7 DO
			pd_ref[i] := G.axis[i].NcToPlc.ActPos - G.init_pos[i];
		END_FOR
	ELSE
		G.program_test_mode := pd_mode;
		G.program_test_status_error_id := 16#7102;
	END_IF
END_IF
IF pd_mode = 0 THEN
	G.program_test_phase := 0;
	G.program_test_sync_state := 0;
	G.program_test_enable := FALSE;
	G.program_test_sample_arm := FALSE;
ELSE
pd_input1 := G.refer[1] + G.init_pos[1];
pd_input2 := G.refer[2] + G.init_pos[2];
IF pd_fault THEN
	pd_state := 12;
	G.program_test_status_error_id := 16#7305;
	IF NOT all_powered THEN
		G.program_test_error_source := 5;
	ELSIF has_axis_error THEN
		G.program_test_error_source := 6;
	ELSIF G.host_comm_timeout THEN
		G.program_test_error_source := 7;
	ELSE
		G.program_test_error_source := 0;
	END_IF
	G.program_test_error_axis := 0;
	G.program_test_error_phase := 0;
	G.program_test_error_target_abs := 0.0;
END_IF
IF G.program_test_abort_req THEN
	G.program_test_abort_req := FALSE;
	pd_state := 11;
END_IF
IF G.experiment_record_overflow THEN
	pd_state := 12;
	G.program_test_status_error_id := 16#7402;
END_IF
FOR i := 1 TO 7 DO
	IF (return_state[i] >= 30) OR (pd_req[i] AND G.return_cmd[i].Done) THEN
		pd_ref[i] := G.axis[i].NcToPlc.ActPos - G.init_pos[i];
	END_IF
	IF pd_req[i] AND G.return_cmd[i].Error THEN
		G.program_test_error_phase := pd_state;
		G.program_test_error_axis := INT_TO_USINT(i);
		G.program_test_error_target_abs := pd_target[i];
		G.program_test_status_error_id := G.return_cmd[i].ErrorId;
		IF G.program_test_status_error_id = 0 THEN
			G.program_test_status_error_id := 16#7306;
		END_IF
		pd_state := 12;
	END_IF
END_FOR
IF (pd_state >= 10) AND G.program_test_setup_req AND pd_all_done AND NOT pd_fault THEN
	pd_state := 0;
	pd_step := 0;
END_IF
IF (pd_state <> 0) AND (pd_state < 10) THEN G.program_test_setup_req := FALSE; END_IF
IF pd_state <> 2 THEN G.program_test_start_req := FALSE; END_IF

pd_baseline_timer(IN:=pd_state = 3, PT:=T#1S);
pd_release_timer(IN:=((pd_state = 1) AND (pd_step = 0)) OR ((pd_state = 5) AND (pd_step = 1)), PT:=pd_release_wait);
pd_reclamp_timer(IN:=(pd_state = 2) OR ((pd_state = 7) AND (pd_step = 1)), PT:=pd_reclamp_wait);
pd_release_lead_timer(IN:=(pd_state = 5) AND (pd_step = 0), PT:=pd_release_lead);
pd_reclamp_lead_timer(IN:=(pd_state = 7) AND (pd_step = 0), PT:=pd_reclamp_lead);
G.program_test_wait_action := 0;

CASE pd_state OF
0:
	IF G.program_test_setup_req AND NOT pd_fault THEN
		G.program_test_setup_req := FALSE;
		G.program_test_start_req := FALSE;
		G.program_test_status_error_id := 0;
		G.program_test_error_source := 0;
		G.program_test_error_axis := 0;
		G.program_test_error_phase := 0;
		G.program_test_error_target_abs := 0.0;
		G.program_test_cycle_index := 0;
		G.program_test_cycle_total := G.program_test_cycle_count;
		G.program_test_setup_done := FALSE;
		pd_ready := FALSE;
		pd_axis := 1;
		IF pd_mode = 2 THEN pd_axis := 6; END_IF
		IF NOT G.self_check_done OR NOT pd_all_done THEN
			G.program_test_status_error_id := 16#7201;
		ELSIF (pd_mode <> 1) AND (pd_mode <> 2) AND (pd_mode <> 4) THEN
			G.program_test_status_error_id := 16#7202;
		ELSIF G.program_test_cycle_count = 0 THEN
			G.program_test_status_error_id := 16#7203;
		ELSIF ((pd_mode = 1) OR (pd_mode = 4)) AND NOT
			((G.program_test_axis1_trigger_from_left_mm >= 0.0) AND
			(G.program_test_axis1_prepare_from_left_mm <= 96.0) AND
			(G.program_test_axis1_prepare_from_left_mm > G.program_test_axis1_trigger_from_left_mm)) THEN
			G.program_test_status_error_id := 16#7204;
		ELSIF (pd_mode = 2) AND NOT
			((G.program_test_axis5_from_left_mm >= 0.0) AND (G.program_test_axis5_from_left_mm <= 670.0) AND
			(G.program_test_axis6_prepare_from_left_mm <= 670.0) AND
			(G.program_test_axis6_trigger_from_left_mm >= 0.0) AND
			(G.program_test_axis6_prepare_from_left_mm > G.program_test_axis6_trigger_from_left_mm)) THEN
			G.program_test_status_error_id := 16#7204;
		ELSIF (pd_mode = 4) AND NOT
			((G.program_test_axis6_prepare_from_left_mm <= 670.0) AND
			(G.program_test_axis6_prepare_from_left_mm -
				UINT_TO_LREAL(G.program_test_cycle_count) *
				(G.program_test_axis1_prepare_from_left_mm - G.program_test_axis1_trigger_from_left_mm) >= 0.0)) THEN
			G.program_test_status_error_id := 16#7204;
		ELSIF NOT ((G.program_test_forward_velocity > 0.0) AND (G.program_test_forward_velocity < 1.0E100) AND
			(G.program_test_forward_acceleration > 0.0) AND (G.program_test_forward_acceleration < 1.0E100) AND
			(G.program_test_forward_deceleration > 0.0) AND (G.program_test_forward_deceleration < 1.0E100) AND
			(G.program_test_forward_jerk > 0.0) AND (G.program_test_forward_jerk < 1.0E100) AND
			(G.program_test_return_velocity > 0.0) AND (G.program_test_return_velocity < 1.0E100) AND
			(G.program_test_return_acceleration > 0.0) AND (G.program_test_return_acceleration < 1.0E100) AND
			(G.program_test_return_deceleration > 0.0) AND (G.program_test_return_deceleration < 1.0E100) AND
			(G.program_test_return_jerk > 0.0) AND (G.program_test_return_jerk < 1.0E100)) THEN
			G.program_test_status_error_id := 16#7205;
		ELSIF (G.program_test_release_wait_ms > 60000) OR (G.program_test_reclamp_wait_ms > 60000) OR
			(G.program_test_release_lead_ms > 60000) OR (G.program_test_reclamp_lead_ms > 60000) THEN
			G.program_test_status_error_id := 16#7207;
		END_IF
		IF G.program_test_status_error_id <> 0 THEN
			pd_state := 12;
		ELSE
			pd_forward.Velocity := G.program_test_forward_velocity;
			pd_forward.Acc := G.program_test_forward_acceleration;
			pd_forward.Dec := G.program_test_forward_deceleration;
			pd_forward.Jerk := G.program_test_forward_jerk;
			pd_return.Velocity := G.program_test_return_velocity;
			pd_return.Acc := G.program_test_return_acceleration;
			pd_return.Dec := G.program_test_return_deceleration;
			pd_return.Jerk := G.program_test_return_jerk;
			pd_release_wait := UDINT_TO_TIME(G.program_test_release_wait_ms);
			pd_reclamp_wait := UDINT_TO_TIME(G.program_test_reclamp_wait_ms);
			pd_release_lead := UDINT_TO_TIME(G.program_test_release_lead_ms);
			pd_reclamp_lead := UDINT_TO_TIME(G.program_test_reclamp_lead_ms);
			pd_open2 := MAX(WORD#5, G.program_test_cylinder2_open_word);
			pd_close2 := MAX(WORD#5, G.program_test_cylinder2_close_word);
			pd_open4 := MAX(WORD#5, G.program_test_cylinder4_open_word);
			pd_close4 := MAX(WORD#5, G.program_test_cylinder4_close_word);
			pd_coupling := G.program_test_cylinder1_coupling_enable OR (pd_mode = 4);
			IF pd_mode = 2 THEN pd_coupling := G.program_test_cylinder3_coupling_enable; END_IF
			G.program_test_target_axis1_abs := G.leftlimit[1] + G.program_test_axis1_prepare_from_left_mm;
			G.program_test_target_axis5_abs := G.leftlimit[5] + G.program_test_axis5_from_left_mm;
			G.program_test_target_axis6_abs := G.leftlimit[6] + G.program_test_axis6_prepare_from_left_mm;
			IF pd_mode = 4 THEN
				// 外源验证两条平移轴使用同一个手柄运动窗口。
				G.program_test_axis6_trigger_from_left_mm :=
					G.program_test_axis6_prepare_from_left_mm -
					(G.program_test_axis1_prepare_from_left_mm - G.program_test_axis1_trigger_from_left_mm);
			END_IF
			G.program_test_target_axis2_deg := G.program_test_axis2_angle_deg;
			G.program_test_target_axis7_deg := G.program_test_axis7_angle_deg;
			FOR i := 1 TO 7 DO
				pd_active[i] := FALSE;
				pd_req[i] := FALSE;
				pd_moved[i] := FALSE;
				pd_ref[i] := G.axis[i].NcToPlc.ActPos - G.init_pos[i];
				pd_target[i] := G.axis[i].NcToPlc.ActPos;
			END_FOR
			IF pd_mode = 2 THEN
				pd_active[5] := TRUE;
				pd_active[6] := TRUE;
				pd_active[7] := TRUE;
				pd_target[5] := G.program_test_target_axis5_abs;
				pd_target[6] := G.program_test_target_axis6_abs;
				pd_target[7] := G.program_test_target_axis7_deg;
				G.program_test_trigger_target_abs := G.leftlimit[6] + G.program_test_axis6_trigger_from_left_mm;
				G.program_test_return_target_abs := pd_target[6];
				G.cylinder3_value := 400;
				IF pd_coupling THEN G.cylinder3_value := 50; END_IF
				G.cylinder4_value := pd_open4;
			ELSE
				pd_active[1] := TRUE;
				pd_active[2] := TRUE;
				pd_target[1] := G.program_test_target_axis1_abs;
				pd_target[2] := G.program_test_target_axis2_deg;
				G.program_test_trigger_target_abs := G.leftlimit[1] + G.program_test_axis1_trigger_from_left_mm;
				G.program_test_return_target_abs := pd_target[1];
				G.cylinder1_value := 400;
				IF pd_coupling THEN G.cylinder1_value := 5; END_IF
				G.cylinder2_value := pd_open2;
			END_IF
			G.program_test_final_target_abs := G.program_test_return_target_abs - G.program_test_final_forward_distance_mm;
			IF pd_mode = 4 THEN
				pd_active[6] := TRUE;
				pd_active[7] := TRUE;
				pd_target[6] := G.program_test_target_axis6_abs;
				pd_target[7] := pd_target[2];
				G.program_test_target_axis7_deg := pd_target[2];
				G.program_test_final_target_abs := G.program_test_return_target_abs;
				G.cylinder3_value := 400;
				G.cylinder4_value := pd_open4;
			END_IF
			pd_state := 1;
		END_IF
	END_IF
1:
	G.program_test_wait_action := 1;
	IF (pd_step = 0) AND pd_release_timer.Q THEN
		FOR i := 1 TO 7 DO pd_req[i] := pd_active[i]; END_FOR
		pd_step := 1;
	END_IF
	IF pd_step = 1 THEN
		G.program_test_wait_action := 0;
		pd_all_done := TRUE;
		FOR i := 1 TO 7 DO
			IF pd_active[i] THEN
				IF G.return_cmd[i].Done THEN
					pd_moved[i] := TRUE;
					pd_req[i] := FALSE;
				END_IF
				IF NOT pd_moved[i] THEN pd_all_done := FALSE; END_IF
			END_IF
		END_FOR
		IF pd_all_done THEN pd_state := 2; END_IF
	END_IF
2:
	IF pd_axis = 1 THEN
		G.cylinder1_value := 400;
		G.cylinder2_value := pd_close2;
	ELSE
		G.cylinder3_value := 400;
		G.cylinder4_value := pd_close4;
	END_IF
	IF pd_mode = 4 THEN G.cylinder4_value := pd_close4; END_IF
	G.program_test_wait_action := 2;
	IF pd_reclamp_timer.Q THEN
		pd_ready := TRUE;
		G.program_test_wait_action := 0;
		IF G.program_test_start_req AND G.experiment_zero_done AND NOT G.experiment_zero_busy THEN
			G.program_test_start_req := FALSE;
			G.program_test_cycle_index := 1;
			pd_state := 3;
		END_IF
	END_IF
3:
	IF pd_baseline_timer.Q THEN pd_state := 4; END_IF
4:
	IF pd_mode = 4 THEN
		IF pd_step = 0 THEN
			pd_anchor1 := G.axis[1].NcToPlc.ActPos;
			pd_anchor5 := G.axis[5].NcToPlc.ActPos;
			pd_anchor6 := G.axis[6].NcToPlc.ActPos;
			G.program_test_handle_cycle := 0;
			pd_step := 1;
		ELSIF G.program_test_handle_cycle = G.program_test_cycle_index THEN
			IF NOT ((pd_input1 >= -1.0E100) AND (pd_input1 <= 1.0E100) AND
				(pd_input2 >= -1.0E100) AND (pd_input2 <= 1.0E100)) THEN
				G.program_test_status_error_id := 16#7208;
				pd_state := 12;
			ELSE
				pd_input1 := LIMIT(G.program_test_trigger_target_abs, pd_input1, G.program_test_return_target_abs);
				pd_ref[1] := pd_input1 - G.init_pos[1];
				pd_ref[2] := pd_input2 - G.init_pos[2];
				pd_ref[5] := G.axis[5].NcToPlc.ActPos - G.init_pos[5];
				pd_ref[6] := pd_anchor6 + pd_input1 - pd_anchor1 - G.init_pos[6];
				pd_ref[7] := pd_input2 - G.init_pos[7];
				IF (pd_input1 <= G.program_test_trigger_target_abs) AND
					(ABS(G.axis[1].NcToPlc.ActPos - G.program_test_trigger_target_abs) <= 0.2) AND
					(ABS(G.axis[5].NcToPlc.ActPos - (pd_ref[5] + G.init_pos[5])) <= 0.2) AND
					(ABS(G.axis[6].NcToPlc.ActPos - (pd_ref[6] + G.init_pos[6])) <= 0.2) AND
					(ABS(G.axis[1].NcToPlc.ActVelo) <= 0.5) AND (ABS(G.axis[6].NcToPlc.ActVelo) <= 0.5) THEN
					pd_state := 5;
				END_IF
			END_IF
		END_IF
	ELSE
		IF pd_step = 0 THEN
			pd_target[pd_axis] := G.program_test_trigger_target_abs;
			pd_req[pd_axis] := TRUE;
			pd_step := 1;
		ELSIF G.return_cmd[pd_axis].Done THEN
			pd_req[pd_axis] := FALSE;
			pd_state := 5;
		END_IF
	END_IF
5:
	G.program_test_wait_action := 1;
	IF pd_axis = 1 THEN
		IF pd_coupling THEN G.cylinder1_value := 5; END_IF
	ELSE
		IF pd_coupling THEN G.cylinder3_value := 50; END_IF
	END_IF
	IF (pd_step = 0) AND (NOT pd_coupling OR pd_release_lead_timer.Q) THEN
		IF pd_axis = 1 THEN G.cylinder2_value := pd_open2; ELSE G.cylinder4_value := pd_open4; END_IF
		pd_step := 1;
	END_IF
	IF (pd_step = 1) AND pd_release_timer.Q THEN pd_state := 6; END_IF
6:
	IF pd_step = 0 THEN
		pd_target[pd_axis] := G.program_test_return_target_abs;
		pd_req[pd_axis] := TRUE;
		pd_step := 1;
	ELSIF G.return_cmd[pd_axis].Done THEN
		pd_req[pd_axis] := FALSE;
		pd_state := 7;
	END_IF
7:
	G.program_test_wait_action := 2;
	IF pd_axis = 1 THEN G.cylinder2_value := pd_close2; ELSE G.cylinder4_value := pd_close4; END_IF
	IF (pd_step = 0) AND (NOT pd_coupling OR pd_reclamp_lead_timer.Q) THEN
		IF pd_axis = 1 THEN G.cylinder1_value := 400; ELSE G.cylinder3_value := 400; END_IF
		pd_step := 1;
	END_IF
	IF (pd_step = 1) AND pd_reclamp_timer.Q THEN pd_state := 8; END_IF
8:
	IF G.program_test_cycle_index < G.program_test_cycle_total THEN
		G.program_test_cycle_index := G.program_test_cycle_index + 1;
		pd_state := 4;
	ELSIF (pd_mode <> 4) AND (G.program_test_final_target_abs < G.program_test_return_target_abs) THEN
		pd_state := 9;
	ELSE
		pd_state := 10;
	END_IF
9:
	IF pd_step = 0 THEN
		pd_target[pd_axis] := G.program_test_final_target_abs;
		pd_req[pd_axis] := TRUE;
		pd_step := 1;
	ELSIF G.return_cmd[pd_axis].Done THEN
		pd_req[pd_axis] := FALSE;
		pd_state := 10;
	END_IF
END_CASE

IF pd_state >= 11 THEN
	pd_ready := FALSE;
	FOR i := 1 TO 7 DO
		pd_req[i] := FALSE;
		IF pd_last_state < 11 THEN pd_ref[i] := G.axis[i].NcToPlc.ActPos - G.init_pos[i]; END_IF
	END_FOR
	G.program_test_start_req := FALSE;
	G.program_test_setup_req := FALSE;
END_IF
IF (pd_mode = 4) AND (pd_state <> 1) AND (pd_state <> 0) THEN
	 pd_ref[7] := pd_ref[2] + G.init_pos[2] - G.init_pos[7];
END_IF

G.program_test_sync_state := 0;
IF (pd_mode = 4) AND (pd_state = 4) THEN
	G.program_test_sync_state := 1;
	IF G.program_test_handle_cycle = G.program_test_cycle_index THEN G.program_test_sync_state := 2; END_IF
ELSIF (pd_mode = 4) AND (pd_state >= 5) AND (pd_state <= 8) THEN
	G.program_test_sync_state := 4;
END_IF
IF pd_state <> 4 THEN G.program_test_handle_cycle := 0; END_IF
FOR i := 1 TO 7 DO
	G.refer[i] := pd_ref[i];
	IF pd_state = 6 THEN
		G.return_cmd[i].Velocity := pd_return.Velocity;
		G.return_cmd[i].Acc := pd_return.Acc;
		G.return_cmd[i].Dec := pd_return.Dec;
		G.return_cmd[i].Jerk := pd_return.Jerk;
	ELSE
		G.return_cmd[i].Velocity := pd_forward.Velocity;
		G.return_cmd[i].Acc := pd_forward.Acc;
		G.return_cmd[i].Dec := pd_forward.Dec;
		G.return_cmd[i].Jerk := pd_forward.Jerk;
	END_IF
	G.return_cmd[i].TargetAbs := pd_target[i];
	G.return_cmd[i].Req := pd_req[i];
END_FOR
G.axis4_fwd_req := FALSE;
G.axis4_rev_req := FALSE;
G.axis1_fast_return := FALSE;
G.axis6_fast_retract := FALSE;
G.startup_smoothing_bypass := FALSE;
G.program_test_phase := pd_state;
G.program_test_enable := (pd_state >= 1) AND (pd_state <= 9);
G.program_test_setup_done := pd_ready;
G.program_test_setup_busy := (pd_state = 1) OR ((pd_state = 2) AND NOT pd_ready);
G.program_test_sample_arm := (pd_state >= 3) AND (pd_state <= 9);
IF (pd_state <> pd_last_state) OR (G.program_test_sync_state <> pd_last_sync) THEN
	G.program_test_event_sequence := G.program_test_event_sequence + 1;
END_IF
IF pd_state <> pd_last_state THEN pd_step := 0; END_IF
pd_last_state := pd_state;
pd_last_sync := G.program_test_sync_state;
END_IF
END_ACTION

ACTION ProgramRecord:

FOR i := 1 TO 2 DO
	IF G.experiment_record_block_ready[i] AND
		(G.experiment_record_block_ack_sequence[i] = G.experiment_record_block_sequence[i]) THEN
		G.experiment_record_block_ready[i] := FALSE;
		G.experiment_record_block_count[i] := 0;
	END_IF
END_FOR
IF G.experiment_record_clear OR G.program_test_sample_clear THEN
	G.experiment_record_clear := FALSE;
	G.program_test_sample_clear := FALSE;
	G.experiment_record_enable := FALSE;
	G.experiment_record_overflow := FALSE;
	G.experiment_record_error_id := 0;
	G.experiment_record_total_count := 0;
	G.program_test_sample_count := 0;
	G.program_test_sample_overflow := FALSE;
	rec_block := 1;
	rec_index := 0;
	rec_sequence := 0;
	rec_was_active := FALSE;
	FOR i := 1 TO 2 DO
		G.experiment_record_block_ready[i] := FALSE;
		G.experiment_record_block_count[i] := 0;
		G.experiment_record_block_sequence[i] := 0;
		G.experiment_record_block_ack_sequence[i] := 16#FFFFFFFF;
	END_FOR
END_IF
IF G.experiment_zero_req THEN
	G.experiment_zero_req := FALSE;
	G.experiment_zero_done := FALSE;
	G.experiment_zero_error_id := 0;
	G.experiment_zero_sample_count := 0;
	G.experiment_zero_busy := pd_ready AND (pd_state = 2) AND NOT pd_fault;
	IF NOT G.experiment_zero_busy THEN G.experiment_zero_error_id := 16#7401; END_IF
	zero_index := 0;
	FOR i := 1 TO 4 DO zero_sum[i] := 0.0; zero_square[i] := 0.0; END_FOR
END_IF
IF G.experiment_zero_busy THEN
	IF pd_fault OR (pd_state <> 2) THEN
		G.experiment_zero_busy := FALSE;
		G.experiment_zero_error_id := 16#7401;
	ELSE
		G.experiment_zero_sample_fn1[zero_index] := G.fn_1_value;
		G.experiment_zero_sample_ft1[zero_index] := G.ft_1_value;
		G.experiment_zero_sample_fn2[zero_index] := G.fn_2_value;
		G.experiment_zero_sample_ft2[zero_index] := G.ft_2_value;
		zero_force[1] := INT_TO_LREAL(G.fn_1_value);
		zero_force[2] := INT_TO_LREAL(G.ft_1_value);
		zero_force[3] := INT_TO_LREAL(G.fn_2_value);
		zero_force[4] := INT_TO_LREAL(G.ft_2_value);
		FOR i := 1 TO 4 DO
			zero_sum[i] := zero_sum[i] + zero_force[i];
			zero_square[i] := zero_square[i] + zero_force[i] * zero_force[i];
		END_FOR
		zero_index := zero_index + 1;
		G.experiment_zero_sample_count := zero_index;
		IF zero_index = 1000 THEN
			FOR i := 1 TO 4 DO
				zero_mean[i] := zero_sum[i] / 1000.0;
				zero_std[i] := SQRT(MAX(0.0, zero_square[i] / 1000.0 - zero_mean[i] * zero_mean[i]));
			END_FOR
			G.experiment_zero_fn1 := zero_mean[1];
			G.experiment_zero_ft1 := zero_mean[2];
			G.experiment_zero_fn2 := zero_mean[3];
			G.experiment_zero_ft2 := zero_mean[4];
			G.experiment_zero_fn1_std := zero_std[1];
			G.experiment_zero_ft1_std := zero_std[2];
			G.experiment_zero_fn2_std := zero_std[3];
			G.experiment_zero_ft2_std := zero_std[4];
			G.experiment_zero_busy := FALSE;
			G.experiment_zero_done := TRUE;
		END_IF
	END_IF
END_IF
rec_capture := G.program_test_sample_arm OR rec_was_active;
rec_was_active := G.program_test_sample_arm;
G.experiment_record_enable := G.program_test_sample_arm AND NOT G.experiment_record_overflow;
IF rec_capture AND NOT G.experiment_record_overflow THEN
IF G.experiment_record_block_ready[rec_block] THEN
	G.experiment_record_overflow := TRUE;
	G.experiment_record_error_id := 16#7402;
	G.experiment_record_enable := FALSE;
	G.program_test_abort_req := TRUE;
ELSE
G.experiment_record_source_mode := pd_mode;
rec_time := UDINT_TO_ULINT(G.experiment_record_total_count) *
	UDINT_TO_ULINT(TwinCAT_SystemInfoVarList._TaskInfo[1].CycleTime) / 10;
rec_sample := MIN(G.program_test_sample_count, UDINT#32767);
G.program_test_sample_index[rec_sample] := G.experiment_record_total_count;
G.program_test_sample_time_us[rec_sample] := rec_time;
G.program_test_sample_phase[rec_sample] := G.program_test_phase;
G.program_test_sample_event_sequence[rec_sample] := G.program_test_event_sequence;
G.program_test_sample_cycle_index[rec_sample] := G.program_test_cycle_index;
G.program_test_sample_sync_state[rec_sample] := G.program_test_sync_state;
G.program_test_sample_axis1_pos[rec_sample] := G.axis[1].NcToPlc.ActPos;
G.program_test_sample_axis1_vel[rec_sample] := G.axis[1].NcToPlc.ActVelo;
G.program_test_sample_axis1_acc[rec_sample] := G.axis[1].NcToPlc.ActAcc;
G.program_test_sample_axis2_pos[rec_sample] := G.axis[2].NcToPlc.ActPos;
G.program_test_sample_axis2_vel[rec_sample] := G.axis[2].NcToPlc.ActVelo;
G.program_test_sample_axis2_acc[rec_sample] := G.axis[2].NcToPlc.ActAcc;
G.program_test_sample_axis5_pos[rec_sample] := G.axis[5].NcToPlc.ActPos;
G.program_test_sample_axis5_vel[rec_sample] := G.axis[5].NcToPlc.ActVelo;
G.program_test_sample_axis5_acc[rec_sample] := G.axis[5].NcToPlc.ActAcc;
G.program_test_sample_axis6_pos[rec_sample] := G.axis[6].NcToPlc.ActPos;
G.program_test_sample_axis6_vel[rec_sample] := G.axis[6].NcToPlc.ActVelo;
G.program_test_sample_axis6_acc[rec_sample] := G.axis[6].NcToPlc.ActAcc;
G.program_test_sample_axis7_pos[rec_sample] := G.axis[7].NcToPlc.ActPos;
G.program_test_sample_axis7_vel[rec_sample] := G.axis[7].NcToPlc.ActVelo;
G.program_test_sample_axis7_acc[rec_sample] := G.axis[7].NcToPlc.ActAcc;
G.program_test_sample_cylinder1[rec_sample] := G.cylinder1_value;
G.program_test_sample_cylinder2[rec_sample] := G.cylinder2_value;
G.program_test_sample_cylinder3[rec_sample] := G.cylinder3_value;
G.program_test_sample_cylinder4[rec_sample] := G.cylinder4_value;
G.program_test_sample_fn1[rec_sample] := G.fn_1_value;
G.program_test_sample_ft1[rec_sample] := G.ft_1_value;
G.program_test_sample_fn2[rec_sample] := G.fn_2_value;
G.program_test_sample_ft2[rec_sample] := G.ft_2_value;
IF G.program_test_sample_count < 32768 THEN
	G.program_test_sample_count := G.program_test_sample_count + 1;
ELSE
	G.program_test_sample_overflow := TRUE;
END_IF
IF rec_block = 1 THEN
	G.experiment_record_block0_index[rec_index] := G.experiment_record_total_count;
	G.experiment_record_block0_time_us[rec_index] := rec_time;
	G.experiment_record_block0_phase[rec_index] := G.program_test_phase;
	G.experiment_record_block0_event_sequence[rec_index] := G.program_test_event_sequence;
	G.experiment_record_block0_cycle_index[rec_index] := G.program_test_cycle_index;
	G.experiment_record_block0_sync_state[rec_index] := G.program_test_sync_state;
	G.experiment_record_block0_axis1_pos[rec_index] := G.axis[1].NcToPlc.ActPos;
	G.experiment_record_block0_axis1_vel[rec_index] := G.axis[1].NcToPlc.ActVelo;
	G.experiment_record_block0_axis1_acc[rec_index] := G.axis[1].NcToPlc.ActAcc;
	G.experiment_record_block0_axis2_pos[rec_index] := G.axis[2].NcToPlc.ActPos;
	G.experiment_record_block0_axis2_vel[rec_index] := G.axis[2].NcToPlc.ActVelo;
	G.experiment_record_block0_axis2_acc[rec_index] := G.axis[2].NcToPlc.ActAcc;
	G.experiment_record_block0_axis5_pos[rec_index] := G.axis[5].NcToPlc.ActPos;
	G.experiment_record_block0_axis5_vel[rec_index] := G.axis[5].NcToPlc.ActVelo;
	G.experiment_record_block0_axis5_acc[rec_index] := G.axis[5].NcToPlc.ActAcc;
	G.experiment_record_block0_axis6_pos[rec_index] := G.axis[6].NcToPlc.ActPos;
	G.experiment_record_block0_axis6_vel[rec_index] := G.axis[6].NcToPlc.ActVelo;
	G.experiment_record_block0_axis6_acc[rec_index] := G.axis[6].NcToPlc.ActAcc;
	G.experiment_record_block0_axis7_pos[rec_index] := G.axis[7].NcToPlc.ActPos;
	G.experiment_record_block0_axis7_vel[rec_index] := G.axis[7].NcToPlc.ActVelo;
	G.experiment_record_block0_axis7_acc[rec_index] := G.axis[7].NcToPlc.ActAcc;
	G.experiment_record_block0_cylinder1[rec_index] := G.cylinder1_value;
	G.experiment_record_block0_cylinder2[rec_index] := G.cylinder2_value;
	G.experiment_record_block0_cylinder3[rec_index] := G.cylinder3_value;
	G.experiment_record_block0_cylinder4[rec_index] := G.cylinder4_value;
	G.experiment_record_block0_fn1[rec_index] := G.fn_1_value;
	G.experiment_record_block0_ft1[rec_index] := G.ft_1_value;
	G.experiment_record_block0_fn2[rec_index] := G.fn_2_value;
	G.experiment_record_block0_ft2[rec_index] := G.ft_2_value;
ELSE
	G.experiment_record_block1_index[rec_index] := G.experiment_record_total_count;
	G.experiment_record_block1_time_us[rec_index] := rec_time;
	G.experiment_record_block1_phase[rec_index] := G.program_test_phase;
	G.experiment_record_block1_event_sequence[rec_index] := G.program_test_event_sequence;
	G.experiment_record_block1_cycle_index[rec_index] := G.program_test_cycle_index;
	G.experiment_record_block1_sync_state[rec_index] := G.program_test_sync_state;
	G.experiment_record_block1_axis1_pos[rec_index] := G.axis[1].NcToPlc.ActPos;
	G.experiment_record_block1_axis1_vel[rec_index] := G.axis[1].NcToPlc.ActVelo;
	G.experiment_record_block1_axis1_acc[rec_index] := G.axis[1].NcToPlc.ActAcc;
	G.experiment_record_block1_axis2_pos[rec_index] := G.axis[2].NcToPlc.ActPos;
	G.experiment_record_block1_axis2_vel[rec_index] := G.axis[2].NcToPlc.ActVelo;
	G.experiment_record_block1_axis2_acc[rec_index] := G.axis[2].NcToPlc.ActAcc;
	G.experiment_record_block1_axis5_pos[rec_index] := G.axis[5].NcToPlc.ActPos;
	G.experiment_record_block1_axis5_vel[rec_index] := G.axis[5].NcToPlc.ActVelo;
	G.experiment_record_block1_axis5_acc[rec_index] := G.axis[5].NcToPlc.ActAcc;
	G.experiment_record_block1_axis6_pos[rec_index] := G.axis[6].NcToPlc.ActPos;
	G.experiment_record_block1_axis6_vel[rec_index] := G.axis[6].NcToPlc.ActVelo;
	G.experiment_record_block1_axis6_acc[rec_index] := G.axis[6].NcToPlc.ActAcc;
	G.experiment_record_block1_axis7_pos[rec_index] := G.axis[7].NcToPlc.ActPos;
	G.experiment_record_block1_axis7_vel[rec_index] := G.axis[7].NcToPlc.ActVelo;
	G.experiment_record_block1_axis7_acc[rec_index] := G.axis[7].NcToPlc.ActAcc;
	G.experiment_record_block1_cylinder1[rec_index] := G.cylinder1_value;
	G.experiment_record_block1_cylinder2[rec_index] := G.cylinder2_value;
	G.experiment_record_block1_cylinder3[rec_index] := G.cylinder3_value;
	G.experiment_record_block1_cylinder4[rec_index] := G.cylinder4_value;
	G.experiment_record_block1_fn1[rec_index] := G.fn_1_value;
	G.experiment_record_block1_ft1[rec_index] := G.ft_1_value;
	G.experiment_record_block1_fn2[rec_index] := G.fn_2_value;
	G.experiment_record_block1_ft2[rec_index] := G.ft_2_value;
END_IF
rec_index := rec_index + 1;
G.experiment_record_total_count := G.experiment_record_total_count + 1;
IF (rec_index = 512) OR NOT G.program_test_sample_arm THEN
	G.experiment_record_block_sequence[rec_block] := rec_sequence;
	G.experiment_record_block_count[rec_block] := INT_TO_UINT(rec_index);
	G.experiment_record_block_ready[rec_block] := TRUE;
	rec_sequence := rec_sequence + 1;
	rec_block := 3 - rec_block;
	rec_index := 0;
END_IF
END_IF
END_IF
END_ACTION

END_FUNCTION_BLOCK

(* stored: Version 1.1.0.1, ProductVersion 3.1.4024.15
   POU handle: Id {687f3d3e-09ee-464b-b8db-c97aea6d31ed}, SpecialFunc None
   Action ProgramDelivery: Id {d90e79ea-aede-41b5-b003-24331ee94001}
   Action ProgramRecord: Id {d90e79ea-aede-41b5-b003-24331ee94002} *)
